# EPICS StreamDevice protocol: docker/PSAppTest/PS_DB_NotSync/tc-l2s_gpio.proto
OutTerminator = CR LF;
InTerminator  = LF;

MaxInput=5;

readDOR {
  out "@DOR?";
  in "%s";
}

readDIR {
  out "@DIR?";
  in "%s";
}

setDOR {
  out "@DO%02u";
  in "@DONE";
  @mismatch{in "@ERR1";}
  @mismatch{in "@ERR2";}
}
